// TIA Portal V17 export
// export: Created 2025-03-07T09:24:28.5150109Z, ExportSetting WithDefaults, DisplayName Totally Integrated Automation Portal, DisplayVersion V17 Update 8, DisplayName TIA Portal Openness, DisplayVersion V17 Update 8, DisplayName TIA Portal Version Control Interface, DisplayVersion V17, DisplayName SINAMICS Startdrive Advanced, DisplayVersion V17 SP2, DisplayName SINAMICS Startdrive G110M, G120, G120C, G120D, G120P, G115D, DisplayVersion V17 SP2, DisplayName SINAMICS Startdrive G130, G150, S120, S150, SINAMICS MV, S210, DisplayVersion V17 SP2, DisplayName STEP 7 Professional, DisplayVersion V17 Update 8, DisplayName SINUMERIK ONE STEP 7 Toolbox, DisplayVersion V17 Update 12, DisplayName SINUMERIK 840D sl STEP 7 Toolbox, DisplayVersion V17 Update 12, DisplayName STEP 7 Safety, DisplayVersion V17 Update 6, DisplayName WinCC Advanced, DisplayVersion V17 Update 8
FUNCTION_BLOCK "FB1013_SAFETY_CLADDING"   // FB1013, F_LAD
{ S7_Optimized_Access := 'TRUE' }
AUTHOR : ETXETAR
VERSION : 1.0
// stored: AutoNumber false, IsIECCheckEnabled false, UDAEnableTagReadback false
   VAR
      F_IEC_Timer_PWR_EN_DEL_2 : TOF;
      F_IEC_Timer_PWR_EN_DEL_3 : TOF;
      F_IEC_Timer_PWR_EN_DEL_4 : TOF;
      F_IEC_Timer_PWR_EN_RES_DEL : TON;
      F_IEC_Timer_PWR_EN_FDBCK : TON;
      F_IEC_Timer_GNTR_DR_FDBCK : TON;
      F_IEC_Timer_FIXT_WRK_COND_FDBCK : TON;
      F_IEC_Timer_MACHINE_E_STOP : TON;
      F_IEC_Timer_CLNT_OFF_01R : TOF;
      F_IEC_Timer_CLNT_OFF_01L : TOF;
      F_IEC_Timer_BIMANUAL_CLOSE : TON;
   END_VAR
   // F_IEC_Timer_PWR_EN_FDBCK.PT := T#30ms;
   // F_IEC_Timer_GNTR_DR_FDBCK.PT := T#30ms;
   // F_IEC_Timer_FIXT_WRK_COND_FDBCK.PT := T#30ms;
   // F_IEC_Timer_MACHINE_E_STOP.PT := T#30ms;
   // F_IEC_Timer_BIMANUAL_CLOSE.PT := T#30ms;
BEGIN

REGION Network 1: *************** EMERGENCY STOP ***************
END_REGION

REGION Network 2: FB E-STOP
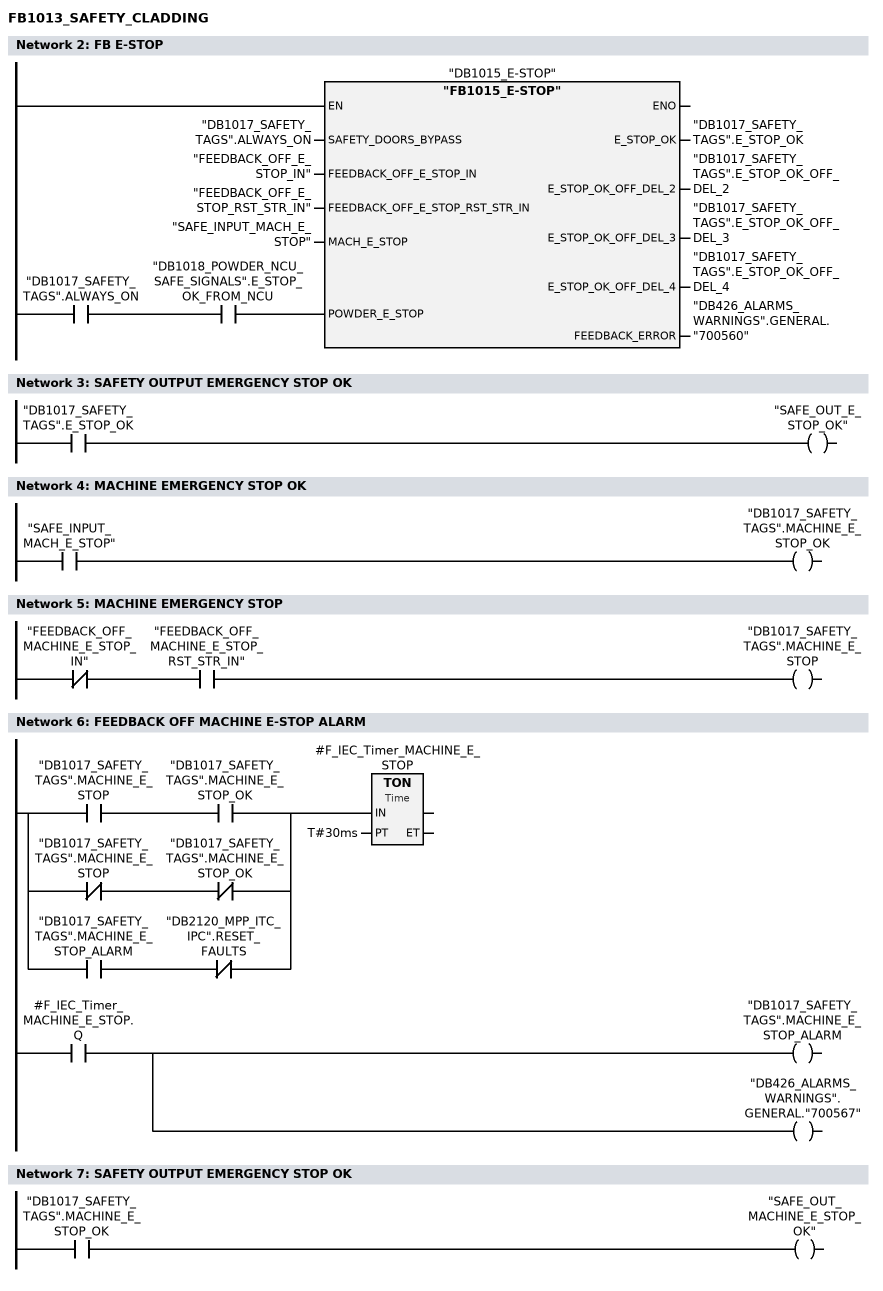
   RUNG wire#powerrail
      "DB1015_E-STOP"(POWDER_E_STOP := wire#w1, SAFETY_DOORS_BYPASS := "DB1017_SAFETY_TAGS".ALWAYS_ON, FEEDBACK_OFF_E_STOP_IN := "FEEDBACK_OFF_E_STOP_IN", FEEDBACK_OFF_E_STOP_RST_STR_IN := "FEEDBACK_OFF_E_STOP_RST_STR_IN", MACH_E_STOP := "SAFE_INPUT_MACH_E_STOP", E_STOP_OK => "DB1017_SAFETY_TAGS".E_STOP_OK, E_STOP_OK_OFF_DEL_2 => "DB1017_SAFETY_TAGS".E_STOP_OK_OFF_DEL_2, E_STOP_OK_OFF_DEL_3 => "DB1017_SAFETY_TAGS".E_STOP_OK_OFF_DEL_3, E_STOP_OK_OFF_DEL_4 => "DB1017_SAFETY_TAGS".E_STOP_OK_OFF_DEL_4, FEEDBACK_ERROR => "DB426_ALARMS_WARNINGS".GENERAL."700560")
   END_RUNG
   RUNG wire#powerrail
      Contact( "DB1017_SAFETY_TAGS".ALWAYS_ON )
      Contact( "DB1018_POWDER_NCU_SAFE_SIGNALS".E_STOP_OK_FROM_NCU )
   END_RUNG wire#w1
   // the same network as SCL:
   "DB1015_E-STOP"(SAFETY_DOORS_BYPASS := "DB1017_SAFETY_TAGS".ALWAYS_ON,   // "FB1015_E-STOP"
                   FEEDBACK_OFF_E_STOP_IN := "FEEDBACK_OFF_E_STOP_IN",
                   FEEDBACK_OFF_E_STOP_RST_STR_IN := "FEEDBACK_OFF_E_STOP_RST_STR_IN",
                   MACH_E_STOP := "SAFE_INPUT_MACH_E_STOP",
                   POWDER_E_STOP := "DB1017_SAFETY_TAGS".ALWAYS_ON AND "DB1018_POWDER_NCU_SAFE_SIGNALS".E_STOP_OK_FROM_NCU,
                   E_STOP_OK => "DB1017_SAFETY_TAGS".E_STOP_OK,
                   E_STOP_OK_OFF_DEL_2 => "DB1017_SAFETY_TAGS".E_STOP_OK_OFF_DEL_2,
                   E_STOP_OK_OFF_DEL_3 => "DB1017_SAFETY_TAGS".E_STOP_OK_OFF_DEL_3,
                   E_STOP_OK_OFF_DEL_4 => "DB1017_SAFETY_TAGS".E_STOP_OK_OFF_DEL_4,
                   FEEDBACK_ERROR => "DB426_ALARMS_WARNINGS".GENERAL."700560");
END_REGION

REGION Network 3: SAFETY OUTPUT EMERGENCY STOP OK
   RUNG wire#powerrail
      Contact( "DB1017_SAFETY_TAGS".E_STOP_OK )
      Coil( "SAFE_OUT_E_STOP_OK" )
   END_RUNG
   // the same network as SCL:
   "SAFE_OUT_E_STOP_OK" := "DB1017_SAFETY_TAGS".E_STOP_OK;
END_REGION

REGION Network 4: MACHINE EMERGENCY STOP OK
   RUNG wire#powerrail
      Contact( "SAFE_INPUT_MACH_E_STOP" )
      Coil( "DB1017_SAFETY_TAGS".MACHINE_E_STOP_OK )
   END_RUNG
   // the same network as SCL:
   "DB1017_SAFETY_TAGS".MACHINE_E_STOP_OK := "SAFE_INPUT_MACH_E_STOP";
END_REGION

REGION Network 5: MACHINE EMERGENCY STOP
   RUNG wire#powerrail
      I_Contact( "FEEDBACK_OFF_MACHINE_E_STOP_IN" )
      Contact( "FEEDBACK_OFF_MACHINE_E_STOP_RST_STR_IN" )
      Coil( "DB1017_SAFETY_TAGS".MACHINE_E_STOP )
   END_RUNG
   // the same network as SCL:
   "DB1017_SAFETY_TAGS".MACHINE_E_STOP := NOT "FEEDBACK_OFF_MACHINE_E_STOP_IN" AND "FEEDBACK_OFF_MACHINE_E_STOP_RST_STR_IN";
END_REGION

REGION Network 6: FEEDBACK OFF MACHINE E-STOP ALARM
   RUNG wire#powerrail
      Contact( "DB1017_SAFETY_TAGS".MACHINE_E_STOP )
      Contact( "DB1017_SAFETY_TAGS".MACHINE_E_STOP_OK )
      wire#w1
      { S7_Templates := "[time_type := Time, codedbool_type := DInt]" } #F_IEC_Timer_MACHINE_E_STOP.TON(pt := T#30ms, et =>)
   END_RUNG
   RUNG wire#powerrail
      I_Contact( "DB1017_SAFETY_TAGS".MACHINE_E_STOP )
      I_Contact( "DB1017_SAFETY_TAGS".MACHINE_E_STOP_OK )
   END_RUNG wire#w1
   RUNG wire#powerrail
      Contact( "DB1017_SAFETY_TAGS".MACHINE_E_STOP_ALARM )
      I_Contact( "DB2120_MPP_ITC_IPC".RESET_FAULTS )
   END_RUNG wire#w1
   RUNG wire#powerrail
      Contact( #F_IEC_Timer_MACHINE_E_STOP.Q )
      wire#w2
      Coil( "DB1017_SAFETY_TAGS".MACHINE_E_STOP_ALARM )
   END_RUNG
   RUNG wire#w2
      Coil( "DB426_ALARMS_WARNINGS".GENERAL."700567" )
   END_RUNG
   // the same network as SCL:
   #F_IEC_Timer_MACHINE_E_STOP.TON(IN := ("DB1017_SAFETY_TAGS".MACHINE_E_STOP AND "DB1017_SAFETY_TAGS".MACHINE_E_STOP_OK) OR (NOT "DB1017_SAFETY_TAGS".MACHINE_E_STOP AND NOT "DB1017_SAFETY_TAGS".MACHINE_E_STOP_OK) OR ("DB1017_SAFETY_TAGS".MACHINE_E_STOP_ALARM AND NOT "DB2120_MPP_ITC_IPC".RESET_FAULTS),
                           PT := T#30ms);
   "DB1017_SAFETY_TAGS".MACHINE_E_STOP_ALARM := #F_IEC_Timer_MACHINE_E_STOP.Q;
   "DB426_ALARMS_WARNINGS".GENERAL."700567" := #F_IEC_Timer_MACHINE_E_STOP.Q;
END_REGION

REGION Network 7: SAFETY OUTPUT EMERGENCY STOP OK
   RUNG wire#powerrail
      Contact( "DB1017_SAFETY_TAGS".MACHINE_E_STOP_OK )
      Coil( "SAFE_OUT_MACHINE_E_STOP_OK" )
   END_RUNG
   // the same network as SCL:
   "SAFE_OUT_MACHINE_E_STOP_OK" := "DB1017_SAFETY_TAGS".MACHINE_E_STOP_OK;
END_REGION
END_FUNCTION_BLOCK
